Fanuc KAREL source: ks00054.KL

PROGRAM KS00054
%STACKSIZE=65535
%PRIORITY=65535
%NOLOCKGROUP
VAR
FLAG : BOOLEAN
N : INTEGER
STATUS : INTEGER
PN : STRING[80]
VN : STRING[80]
-- UNRESOLVED DECLARATIONS (source type spelling not recovered)
-- A : ARRAY[4] OF TYPE_0x1100 (type_u16=0x3100)
-- B : ARRAY[4] OF TYPE_0x1100 (type_u16=0x3100)
BEGIN
PN=''
VN='A'
-- UNSAFE_SOURCE_IR line 19: N = native_s16_value(A)
END KS00054
